// Mitsubishi GX Works2 project: 0703-공개문제20   PLC: Q02/Q02H

PROGRAM MAIN
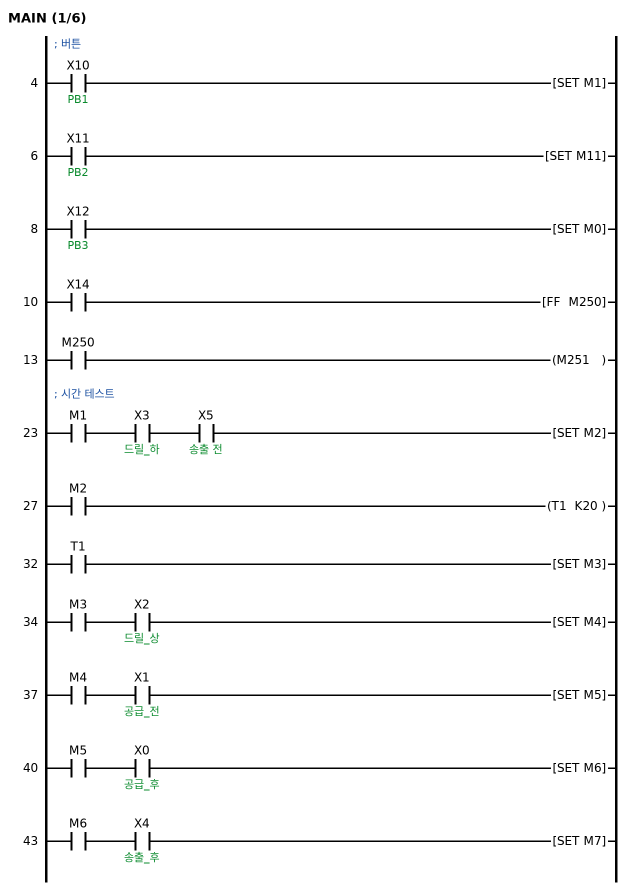
; 버튼
4     LD      X10  ; PB1
      SET     M1
6     LD      X11  ; PB2
      SET     M11
8     LD      X12  ; PB3
      SET     M0
10    LD      X14
      FF      M250
13    LD      M250
      OUT     M251
; 시간 테스트
23    LD      M1
      AND     X3  ; 드릴_하
      AND     X5  ; 송출 전
      SET     M2
27    LD      M2
      OUT     T1 K20
32    LD      T1
      SET     M3
34    LD      M3
      AND     X2  ; 드릴_상
      SET     M4
37    LD      M4
      AND     X1  ; 공급_전
      SET     M5
40    LD      M5
      AND     X0  ; 공급_후
      SET     M6
43    LD      M6
      AND     X4  ; 송출_후
      SET     M7
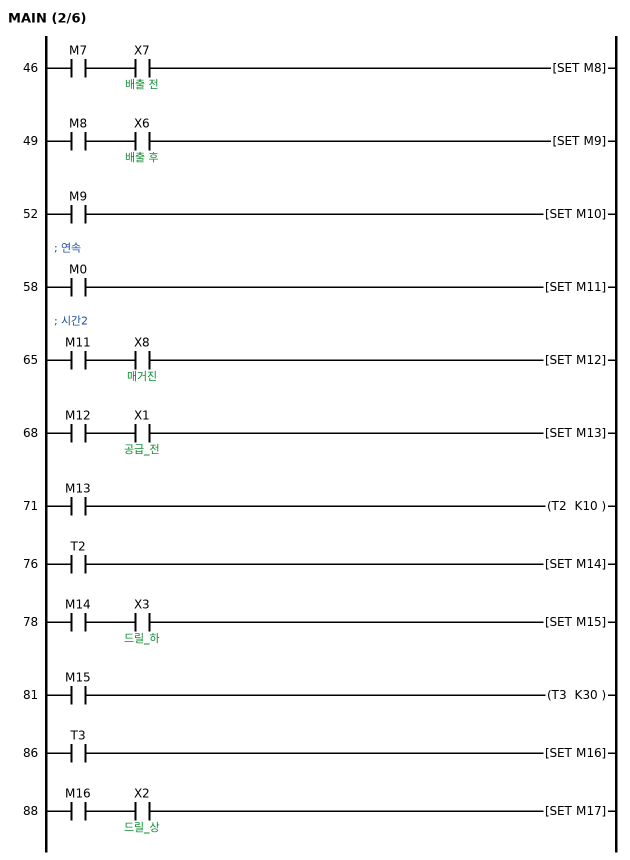
46    LD      M7
      AND     X7  ; 배출 전
      SET     M8
49    LD      M8
      AND     X6  ; 배출 후
      SET     M9
52    LD      M9
      SET     M10
; 연속
58    LD      M0
      SET     M11
; 시간2
65    LD      M11
      AND     X8  ; 매거진
      SET     M12
68    LD      M12
      AND     X1  ; 공급_전
      SET     M13
71    LD      M13
      OUT     T2 K10
76    LD      T2
      SET     M14
78    LD      M14
      AND     X3  ; 드릴_하
      SET     M15
81    LD      M15
      OUT     T3 K30
86    LD      T3
      SET     M16
88    LD      M16
      AND     X2  ; 드릴_상
      SET     M17
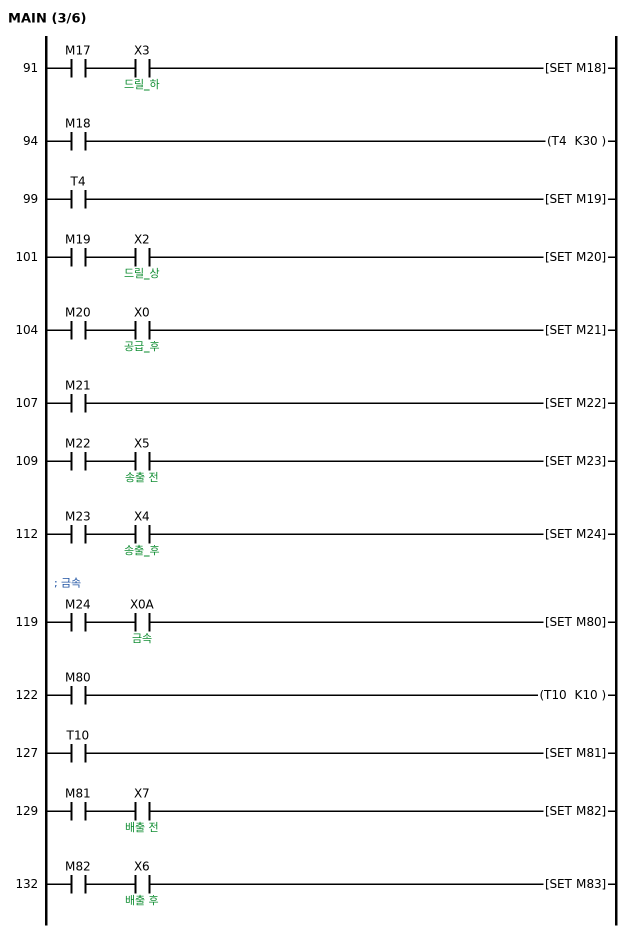
91    LD      M17
      AND     X3  ; 드릴_하
      SET     M18
94    LD      M18
      OUT     T4 K30
99    LD      T4
      SET     M19
101   LD      M19
      AND     X2  ; 드릴_상
      SET     M20
104   LD      M20
      AND     X0  ; 공급_후
      SET     M21
107   LD      M21
      SET     M22
109   LD      M22
      AND     X5  ; 송출 전
      SET     M23
112   LD      M23
      AND     X4  ; 송출_후
      SET     M24
; 금속
119   LD      M24
      AND     X0A  ; 금속
      SET     M80
122   LD      M80
      OUT     T10 K10
127   LD      T10
      SET     M81
129   LD      M81
      AND     X7  ; 배출 전
      SET     M82
132   LD      M82
      AND     X6  ; 배출 후
      SET     M83
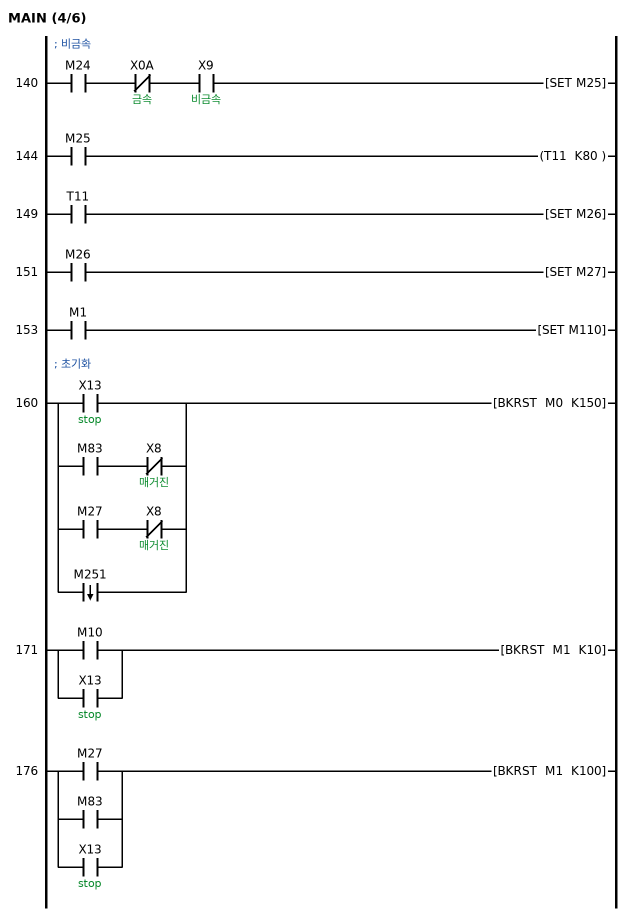
; 비금속
140   LD      M24
      ANI     X0A  ; 금속
      AND     X9  ; 비금속
      SET     M25
144   LD      M25
      OUT     T11 K80
149   LD      T11
      SET     M26
151   LD      M26
      SET     M27
153   LD      M1
      SET     M110
; 초기화
160   LD      X13  ; stop
      LD      M83
      ANI     X8  ; 매거진
      ORB
      LD      M27
      ANI     X8  ; 매거진
      ORB
      ORF     M251
      BKRST   M0 K150
171   LD      M10
      OR      X13  ; stop
      BKRST   M1 K10
176   LD      M27
      OR      M83
      OR      X13  ; stop
      BKRST   M1 K100
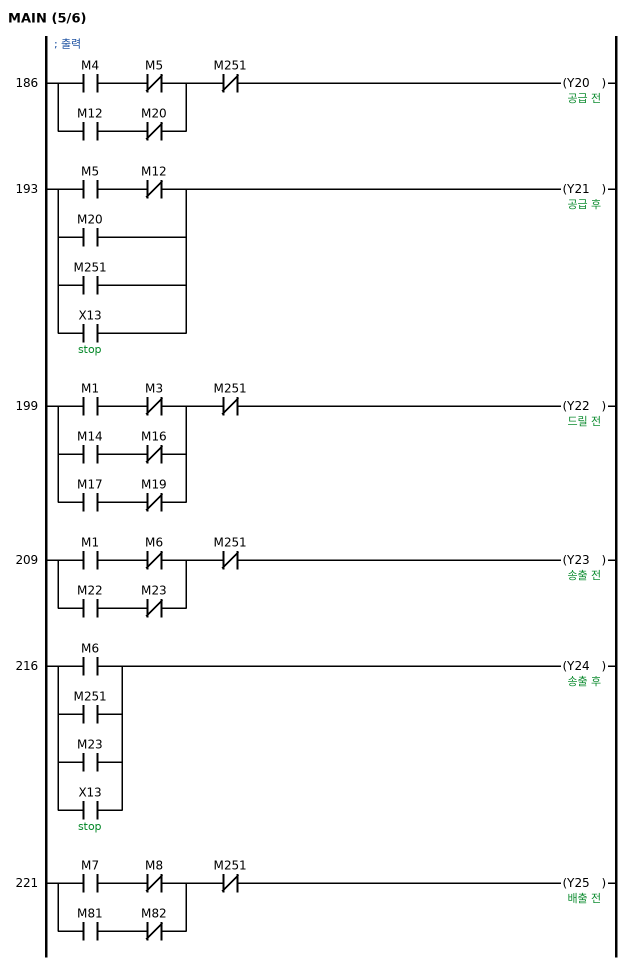
; 출력
186   LD      M4
      ANI     M5
      LD      M12
      ANI     M20
      ORB
      ANI     M251
      OUT     Y20  ; 공급 전
193   LD      M5
      ANI     M12
      OR      M20
      OR      M251
      OR      X13  ; stop
      OUT     Y21  ; 공급 후
199   LD      M1
      ANI     M3
      LD      M14
      ANI     M16
      ORB
      LD      M17
      ANI     M19
      ORB
      ANI     M251
      OUT     Y22  ; 드릴 전
209   LD      M1
      ANI     M6
      LD      M22
      ANI     M23
      ORB
      ANI     M251
      OUT     Y23  ; 송출 전
216   LD      M6
      OR      M251
      OR      M23
      OR      X13  ; stop
      OUT     Y24  ; 송출 후
221   LD      M7
      ANI     M8
      LD      M81
      ANI     M82
      ORB
      ANI     M251
      OUT     Y25  ; 배출 전
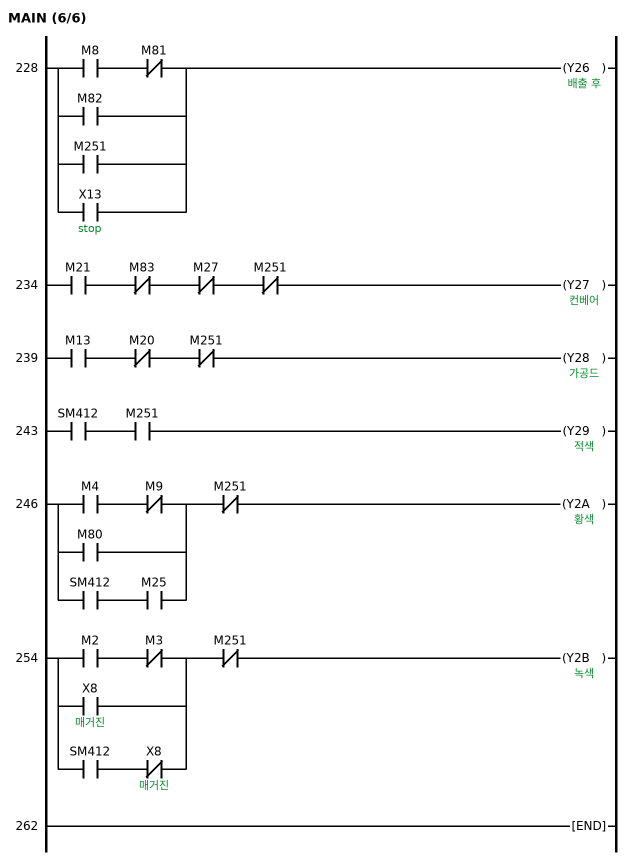
228   LD      M8
      ANI     M81
      OR      M82
      OR      M251
      OR      X13  ; stop
      OUT     Y26  ; 배출 후
234   LD      M21
      ANI     M83
      ANI     M27
      ANI     M251
      OUT     Y27  ; 컨베어
239   LD      M13
      ANI     M20
      ANI     M251
      OUT     Y28  ; 가공드
243   LD      SM412
      AND     M251
      OUT     Y29  ; 적색
246   LD      M4
      ANI     M9
      OR      M80
      LD      SM412
      AND     M25
      ORB
      ANI     M251
      OUT     Y2A  ; 황색
254   LD      M2
      ANI     M3
      OR      X8  ; 매거진
      LD      SM412
      ANI     X8  ; 매거진
      ORB
      ANI     M251
      OUT     Y2B  ; 녹색
262   END
END_PROGRAM

PROGRAM MAIN1
0     END
END_PROGRAM
